Fanuc KAREL source: kt00012.KL

-- PROVISIONAL review KL for V940-1; original PC SHA256 fb7fe349e2ca8797864953866d4ba01e3fe81edf3f40e411e29665465c0b4d87
-- Incomplete behavior may be omitted. Consult companion uncertainty JSON. Do not deploy.
PROGRAM KT00012
%NOLOCKGROUP
VAR
  R1 : REAL
  R2 : REAL
  OUT : REAL
BEGIN
  -- V9_ZERO_TABLE_METADATA_HINT layout=0001; no indexed target words; source/name/runtime held
  -- UNRESOLVED_PC offsets 5-16; opcodes 2E,23
  -- UNRESOLVED_PC offsets 21-32; opcodes 2E,23
  -- UNRESOLVED_PC offsets 37-48; opcodes 2E,23
  -- UNRESOLVED_PC offsets 53-64; opcodes 2E,23
  -- UNRESOLVED_PC offsets 69-88; opcodes 21,21,69,23
  -- UNRESOLVED_PC offsets 93-97; opcodes 7F
END KT00012
